{attribute 'GeneratedUsingTerminal: EK1960-2600-0021'}
{attribute addProperty BoxType "EK1960-2600-0021"}
{attribute addProperty Id "EtcSlaveTerminalBaseModule_1_FSoEModule_1_FSoE_B78AD590104Module_2_FSOUTModule_2_FSOUT_E84B1B0028Module_3_FSLOGICModule_3_FSLOGIC_DEAB45222WcStateAT %I*WcState_B516A2644InfoDataAT %I*InfoData_32EB74EA10"}
{attribute addProperty CRC "2806305696"}
{attribute addProperty Size "148"}
TYPE EK1960_A744D3A0 EXTENDS EtcSlaveTerminalBase :
STRUCT
	{attribute addProperty Name "Module_1_FSoE"}
	Module_1_FSoE : Module_1_FSoE_B78AD590;
	{attribute addProperty Name "Module_2_FSOUT"}
	Module_2_FSOUT : Module_2_FSOUT_E84B1B00;
	{attribute addProperty Name "Module_3_FSLOGIC"}
	Module_3_FSLOGIC : Module_3_FSLOGIC_DEAB4522;
	{attribute addProperty Name "WcState"}
	WcState : WcState_B516A264;
	{attribute addProperty Name "InfoData"}
	InfoData : InfoData_32EB74EA;
END_STRUCT
END_TYPE

(* stored: Version 1.2.0.0, ProductVersion 3.1.4024.9
   DUT EK1960_A744D3A0: Id {ab9fa537-7e66-4516-905c-1dba9f96f7ec} *)
